FUNCTION_BLOCK Gripper2Ctrl (* Basic Function Block Type *)
  (* Standard: 61499-2 *)
  (* Version 0.0, 3/23/2016, Aalto_IT, nxtControl GmbH, Template *)
  PACKAGE Main;
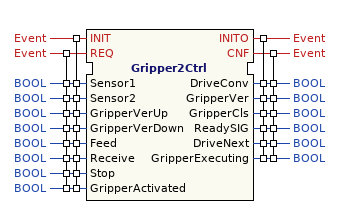
  EVENT_INPUT
    INIT WITH Sensor1, Sensor2, GripperVerUp, GripperVerDown, Feed, Receive, Stop, GripperActivated; (* Initialization Request *)
    REQ WITH Sensor1, Sensor2, GripperVerUp, GripperVerDown, Feed, Receive, Stop, GripperActivated; (* Normal Execution Request *)
  END_EVENT
  EVENT_OUTPUT
    INITO WITH DriveConv, GripperVer, GripperCls, ReadySIG, DriveNext, GripperExecuting; (* Initialization Confirm *)
    CNF WITH DriveConv, GripperVer, GripperCls, ReadySIG, DriveNext, GripperExecuting; (* Execution Confirmation *)
  END_EVENT
  VAR_INPUT
    Sensor1 : BOOL; (* Input event qualifier *)
    Sensor2 : BOOL;
    GripperVerUp : BOOL;
    GripperVerDown : BOOL;
    Feed : BOOL;
    Receive : BOOL;
    Stop : BOOL;
    GripperActivated : BOOL;
  END_VAR
  VAR_OUTPUT
    DriveConv : BOOL; (* Output event qualifier *)
    GripperVer : BOOL;
    GripperCls : BOOL;
    ReadySIG : BOOL;
    DriveNext : BOOL;
    GripperExecuting : BOOL;
  END_VAR
  VAR
    TimeStamp : DATE_AND_TIME;
  END_VAR
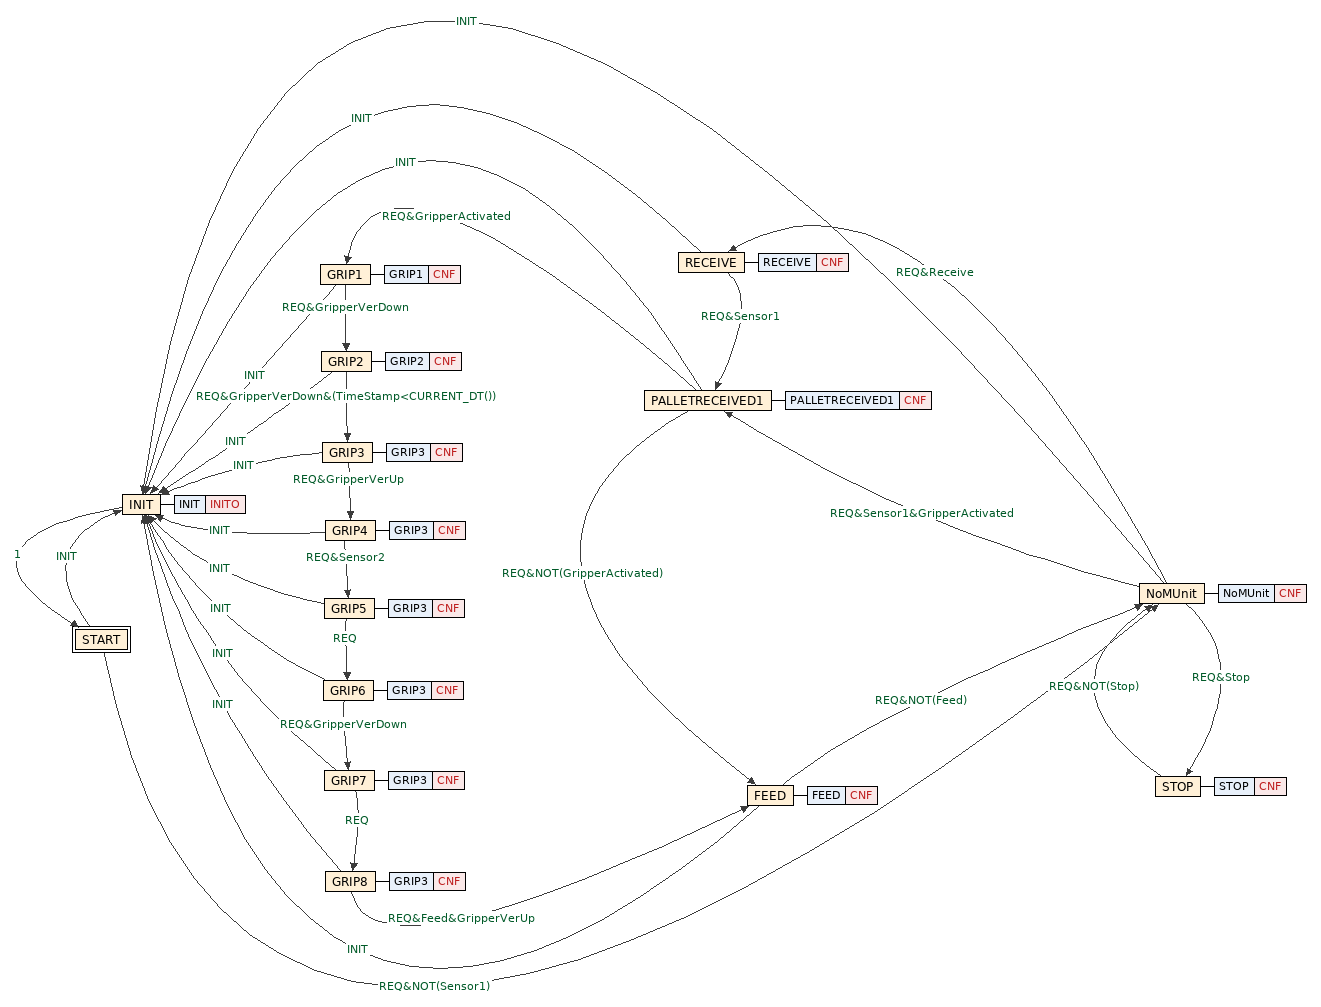
  EC_STATES
    START; (* Initial State *)
    INIT : INIT -> INITO; (* Initialization *)
    NoMUnit : NoMUnit -> CNF;
    PALLETRECEIVED1 : PALLETRECEIVED1 -> CNF;
    GRIP1 : GRIP1 -> CNF;
    GRIP2 : GRIP2 -> CNF;
    GRIP3 : GRIP3 -> CNF;
    GRIP4 : GRIP3 -> CNF;
    FEED : FEED -> CNF;
    GRIP5 : GRIP3 -> CNF;
    GRIP6 : GRIP3 -> CNF;
    GRIP7 : GRIP3 -> CNF;
    GRIP8 : GRIP3 -> CNF;
    RECEIVE : RECEIVE -> CNF;
    STOP : STOP -> CNF;
  END_STATES
  EC_TRANSITIONS
    NoMUnit TO PALLETRECEIVED1 := REQ&Sensor1&GripperActivated;
    PALLETRECEIVED1 TO GRIP1 := REQ&GripperActivated;
    GRIP1 TO GRIP2 := REQ&GripperVerDown;
    GRIP2 TO GRIP3 := REQ&GripperVerDown&(TimeStamp<CURRENT_DT());
    GRIP3 TO GRIP4 := REQ&GripperVerUp;
    GRIP8 TO FEED := REQ&Feed&GripperVerUp;
    FEED TO NoMUnit := REQ&NOT(Feed);
    GRIP7 TO GRIP8 := REQ;
    GRIP6 TO GRIP7 := REQ&GripperVerDown;
    GRIP5 TO GRIP6 := REQ;
    GRIP4 TO GRIP5 := REQ&Sensor2;
    PALLETRECEIVED1 TO FEED := REQ&NOT(GripperActivated);
    NoMUnit TO RECEIVE := REQ&Receive;
    RECEIVE TO PALLETRECEIVED1 := REQ&Sensor1;
    GRIP8 TO INIT := INIT;
    GRIP7 TO INIT := INIT;
    GRIP6 TO INIT := INIT;
    GRIP5 TO INIT := INIT;
    GRIP4 TO INIT := INIT;
    GRIP3 TO INIT := INIT;
    GRIP2 TO INIT := INIT;
    GRIP1 TO INIT := INIT;
    RECEIVE TO INIT := INIT;
    FEED TO INIT := INIT;
    PALLETRECEIVED1 TO INIT := INIT;
    NoMUnit TO INIT := INIT;
    STOP TO NoMUnit := REQ&NOT(Stop);
    NoMUnit TO STOP := REQ&Stop;
    INIT TO START := 1;
    START TO INIT := INIT;
    START TO NoMUnit := REQ&NOT(Sensor1);
  END_TRANSITIONS
  ALGORITHM INIT IN ST: (* Initialization algorithm *)
DriveConv:=0;
GripperVer:=0;
GripperCls:=0;
DriveNext:=0;
ReadySIG:=1;
GripperExecuting:=0;
  END_ALGORITHM
  ALGORITHM REQ IN ST: (* Normally executed algorithm *)
;
  END_ALGORITHM
  ALGORITHM NoMUnit IN ST:
DriveConv:=0;
GripperVer:=0;
GripperCls:=0;
ReadySIG:=1;
DriveNext:=0;
  END_ALGORITHM
  ALGORITHM PALLETRECEIVED1 IN ST:
DriveConv:=0;
GripperVer:=0;
GripperCls:=0;
ReadySIG:=0;
DriveNext:=0;
  END_ALGORITHM
  ALGORITHM GRIP1 IN ST:
DriveConv:=0;
GripperVer:=1;
GripperCls:=0;
ReadySIG:=0;
DriveNext:=0;
GripperExecuting:=1;
  END_ALGORITHM
  ALGORITHM GRIP2 IN ST:
DriveConv:=0;
GripperVer:=1;
GripperCls:=1;
ReadySIG:=0;
TimeStamp:=ADD_DT_TIME(CURRENT_DT(),T#0.5s);
DriveNext:=0;
  END_ALGORITHM
  ALGORITHM GRIP3 IN ST:
DriveConv:=0;
GripperVer:=0;
GripperCls:=1;
ReadySIG:=0;
DriveNext:=0;
  END_ALGORITHM
  ALGORITHM FEED IN ST:
DriveConv:=1;
GripperVer:=0;
GripperCls:=0;
ReadySIG:=0;
DriveNext:=1;
  END_ALGORITHM
  ALGORITHM GRIP6 IN ST:
DriveConv:=0;
GripperVer:=1;
GripperCls:=1;
ReadySIG:=0;
DriveNext:=0;
  END_ALGORITHM
  ALGORITHM GRIP7 IN ST:
DriveConv:=0;
GripperVer:=1;
GripperCls:=0;
ReadySIG:=0;
DriveNext:=0;
  END_ALGORITHM
  ALGORITHM GRIP8 IN ST:
DriveConv:=0;
GripperVer:=0;
GripperCls:=0;
ReadySIG:=0;
DriveNext:=0;
GripperExecuting:=0;
  END_ALGORITHM
  ALGORITHM NOPALLET1 IN ST:
DriveConv:=0;
GripperVer:=0;
GripperCls:=1;
ReadySIG:=1;
DriveNext:=0;
  END_ALGORITHM
  ALGORITHM PALLETRECEIVED IN ST:
DriveConv:=0;
GripperVer:=0;
GripperCls:=0;
ReadySIG:=0;
DriveNext:=0;
  END_ALGORITHM
  ALGORITHM RECEIVE IN ST:
DriveConv:=1;
GripperVer:=0;
GripperCls:=0;
ReadySIG:=1;
DriveNext:=0;
  END_ALGORITHM
  ALGORITHM FEED1 IN ST:
DriveConv:=1;
GripperVer:=0;
GripperCls:=1;
ReadySIG:=0;
DriveNext:=1;
  END_ALGORITHM
  ALGORITHM RECEIVE1 IN ST:
DriveConv:=1;
GripperVer:=0;
GripperCls:=1;
ReadySIG:=1;
DriveNext:=0;
  END_ALGORITHM
  ALGORITHM STOP IN ST:
DriveConv:=0;
GripperVer:=0;
GripperCls:=0;
DriveNext:=0;
ReadySIG:=0;
  END_ALGORITHM
END_FUNCTION_BLOCK
